FUNCTION_BLOCK PML_Method_Base IMPLEMENTS I_Cyclic
VAR_INPUT
END_VAR
VAR_OUTPUT
END_VAR
VAR
	ipackml : IPmlStateMachine;
END_VAR

{analysis -2}

METHOD PROTECTED Aborted : BOOL
VAR_INPUT
END_VAR
Aborted := true;
END_METHOD

METHOD PROTECTED Aborting : BOOL
VAR_INPUT
END_VAR
ipackml.SetStateComplete();
Aborting := TRUE;
END_METHOD

METHOD PROTECTED Clearing : BOOL
VAR_INPUT
END_VAR
ipackml.SetStateComplete();
Clearing := TRUE;
END_METHOD

METHOD PROTECTED Completed : BOOL
VAR_INPUT
END_VAR
Completed := TRUE;
END_METHOD

METHOD PROTECTED Completing : BOOL
VAR_INPUT
END_VAR
ipackml.SetStateComplete();
Completing := TRUE;
END_METHOD

METHOD PUBLIC Cycle : HRESULT
VAR
	StateCallResult : BOOL;
END_VAR
CASE ipackml.GetCurrentState() OF
	E_PMLState.ePMLState_Clearing:
		StateCallResult := Clearing();
	E_PMLState.ePMLState_Aborted:
		StateCallResult := Aborted();
	E_PMLState.ePMLState_Aborting:
		StateCallResult := Aborting();
	E_PMLState.ePMLState_Complete:
		StateCallResult := Completed();
	E_PMLState.ePMLState_Completing:
		StateCallResult := Completing();
	E_PMLState.ePMLState_Execute:
		StateCallResult := Execute();
	E_PMLState.ePMLState_Held:
		StateCallResult := Held();
	E_PMLState.ePMLState_Holding:
		StateCallResult := Holding();
	E_PMLState.ePMLState_Idle:
		StateCallResult := Idle();
	E_PMLState.ePMLState_Resetting:
		StateCallResult := Resetting();
	E_PMLState.ePMLState_Starting:
		StateCallResult := Starting();
	E_PMLState.ePMLState_Stopped:
		StateCallResult := Stopped();
	E_PMLState.ePMLState_Stopping:
		StateCallResult := Stopping();
	E_PMLState.ePMLState_Suspended:
		StateCallResult := Suspended();
	E_PMLState.ePMLState_Suspending:
		StateCallResult := Suspending();
	E_PMLState.ePMLState_Undefined:
		StateCallResult := Undefined();
	E_PMLState.ePMLState_Unholding:
		StateCallResult := Unholding();
	E_PMLState.ePMLState_Unsuspending:
		StateCallResult := Unsuspending();
	ELSE
		Cycle := E_FAIL;
END_CASE
IF StateCallResult THEN
	Cycle := S_OK;
ELSE
	Cycle := E_FAIL;
END_IF
END_METHOD

METHOD PROTECTED Execute : BOOL
VAR_INPUT
END_VAR
Execute := true;
END_METHOD

METHOD PROTECTED Held : BOOL
VAR_INPUT
END_VAR
Held := TRUE;
END_METHOD

METHOD PROTECTED Holding : BOOL
VAR_INPUT
END_VAR
ipackml.SetStateComplete();
Holding := TRUE;
END_METHOD

METHOD PROTECTED Idle : BOOL
VAR_INPUT
END_VAR
Idle := TRUE;
END_METHOD

PROPERTY PUBLIC PackMLStateMachine : IPmlStateMachine
GET
PackMLStateMachine := ipackml;
END_GET
SET
ipackml := PackMLStateMachine;
END_SET
END_PROPERTY

METHOD PROTECTED Resetting : BOOL
VAR_INPUT
END_VAR
ipackml.SetStateComplete();
Resetting := TRUE;
END_METHOD

METHOD PROTECTED Starting : BOOL
VAR_INPUT
END_VAR
ipackml.SetStateComplete();
Starting := TRUE;
END_METHOD

METHOD PROTECTED Stopped : BOOL
VAR_INPUT
END_VAR
Stopped := TRUE;
END_METHOD

METHOD PROTECTED Stopping : BOOL
VAR_INPUT
END_VAR
ipackml.SetStateComplete();
Stopping := TRUE;
END_METHOD

METHOD PROTECTED Suspended : BOOL
VAR_INPUT
END_VAR
Suspended := TRUE;
END_METHOD

METHOD PROTECTED Suspending : BOOL
VAR_INPUT
END_VAR
ipackml.SetStateComplete();
Suspending := TRUE;
END_METHOD

METHOD PROTECTED Undefined : BOOL
VAR_INPUT
END_VAR
Undefined := TRUE;
END_METHOD

METHOD PROTECTED Unholding : BOOL
VAR_INPUT
END_VAR
ipackml.SetStateComplete();
Unholding := TRUE;
END_METHOD

METHOD PROTECTED Unsuspending : BOOL
VAR_INPUT
END_VAR
ipackml.SetStateComplete();
Unsuspending := TRUE;
END_METHOD

END_FUNCTION_BLOCK

(* stored: Version 1.1.0.1
   POU PML_Method_Base: Id {44604a6d-2a49-42c2-9e01-3b91f586bd10}, SpecialFunc None
   Folder Action_States: Id {7719f547-9feb-4937-b59c-20a931e8ad41}
   Folder Wait_States: Id {2c32ef48-514a-481f-8d0d-8b942ec72232}
   Method Aborted: Id {3a7a888a-3488-4e5a-a007-83e4c843c99f}
   Method Aborting: Id {8eff91aa-7f1e-4fd3-a545-3f5a7ea2c597}
   Method Clearing: Id {64009759-9dcd-45d2-8a6f-25e2864a6e21}
   Method Completed: Id {8db612cd-d25e-4f0e-8127-a16fd256f153}
   Method Completing: Id {6703021e-8530-4771-aaae-3cde4b26799f}
   Method Cycle: Id {63d4d0a3-0b0d-4da4-b46f-2e93b903d4c3}
   Method Execute: Id {5484d7e2-b3e2-4d00-adc7-910112ca7207}
   Method Held: Id {004fe5f5-1493-4831-9660-53dd53b37151}
   Method Holding: Id {5db35954-b6c7-44bc-be52-fc73d3a1d8dd}
   Method Idle: Id {8dbd11b2-5cb0-447d-943f-09b5ebac915e}
   Property PackMLStateMachine: Id {1848e61a-7da6-4ad1-b602-39cdcadd7b88}
   Get Get: Id {70e77818-fff6-4ea3-a9c0-c213ac8f42fa}
   Set Set: Id {460c6705-7754-439c-980c-6919cb3d2d7b}
   Method Resetting: Id {e31b868e-5e8d-487c-b4ed-f6356e1fe4b9}
   Method Starting: Id {98960e70-b46e-4571-b670-dbf1d87ceb4e}
   Method Stopped: Id {1e2bcc54-c534-460e-a757-8d619b18aa64}
   Method Stopping: Id {b994c5a8-ad42-4f18-9920-c355d4106f0a}
   Method Suspended: Id {23225890-9944-4ad7-8f64-13b40599a318}
   Method Suspending: Id {aec63dc9-e7be-4fa6-bc82-be2d206971e8}
   Method Undefined: Id {4f5c025e-6f39-48a9-b127-9303fab086d4}
   Method Unholding: Id {3d0e100d-fc99-4eff-854c-988cbc39a6e1}
   Method Unsuspending: Id {5ce0470e-2c5c-47a1-b247-b5084620a760} *)
